Universal Robots PolyScope program: industrial_CHAIYO_TURBO.urp

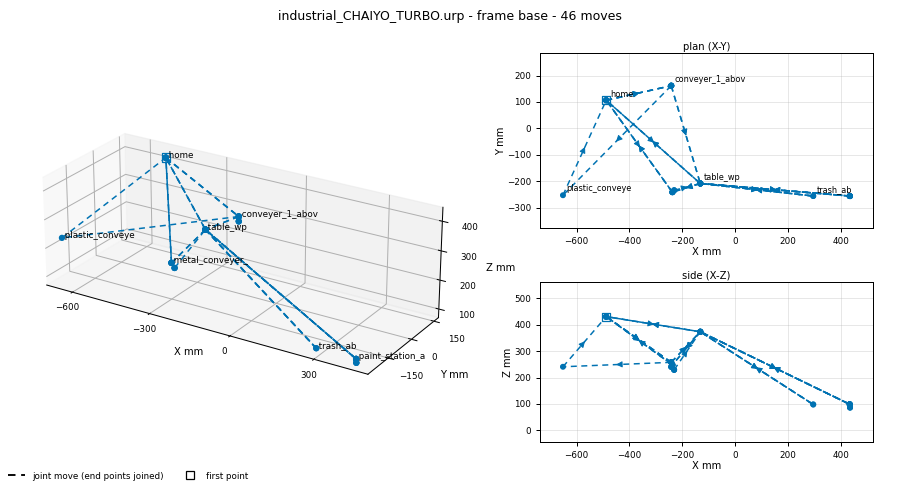
[picture p0: tool path of industrial_CHAIYO_TURBO.urp in frame base, 46 of 46 moves have a stored position in this frame; points joined in program order, loops and branches not executed]
Program industrial_CHAIYO_TURBO (createdIn=3.3.2.266 lastSavedIn=3.3.2.266 directory=/programs/usbdisk installation=default robotSerialNumber=2016353468)
Calibrated DH parameters: a=[0.000201, -0.204825, -0.377339, 0.000067, 0.000035, 0]; d=[0.089016, 277.403916, -258.203358, -19.0904, 0.094913, 0.082586]; alpha=[1.570161, 0.001342, -0.005575, 1.569994, -1.570842, 0]; deltaTheta=[0.000008, 1.067914, -1.344269, 0.276418, -0.000094, 0.00004]
Robot Program (runOnlyOnce=false motionType=MoveJ speed=1.047198 acceleration=1.396263 recalculateMotions=false)
  Set DigitalOutput pin=digital_out[4]; digitalValue=0
  var_1 := 0
  var_2 := 0
  var_3 := 0
  MoveJ speed 30 deg/s, acceleration 50 deg/s^2 (recalculateMotions=false)
    Waypoint home: TCP in base x=-488.151 y=106.291 z=430.627 mm, rx=1.1928 ry=2.9028 rz=-0.0084 rad; joints [180.494, -90.027, -89.995, -90.031, 90.023, -45] deg
  Wait DigitalInput pin=digital_in[0]; digitalValue=1
  If digital_in[1]
    var_1 := 1
  If digital_in[2]
    var_2 := 1
  If digital_in[3]
    var_3 := 1
  Set DigitalOutput pin=digital_out[0]; digitalValue=1
  Set DigitalOutput pin=digital_out[1]; digitalValue=1
  Switch expression=var_1*4+var_2*2+var_3*1
    Case (caseValue=1)
      MoveJ speed 50 deg/s, acceleration 60 deg/s^2 (recalculateMotions=false)
        Waypoint conveyer_1_abov: TCP in base x=-241.88 y=161.267 z=257.494 mm, rx=1.1929 ry=2.9028 rz=-0.0085 rad; joints [168.609, -62.296, -136.212, -71.617, 90.039, -56.942] deg
        Set DigitalOutput pin=digital_out[4]; digitalValue=1
      MoveJ speed 10 deg/s, acceleration 20 deg/s^2 (recalculateMotions=false)
        Waypoint conveyer_1: TCP in base x=-241.869 y=161.248 z=240.365 mm, rx=1.1929 ry=2.9028 rz=-0.0085 rad; joints [168.613, -63.476, -138.325, -68.325, 90.05, -56.955] deg
        Waypoint conveyer_1_abov: TCP in base x=-241.88 y=161.267 z=257.494 mm, rx=1.1929 ry=2.9028 rz=-0.0085 rad; joints [168.609, -62.296, -136.212, -71.617, 90.039, -56.942] deg
      MoveJ speed 50 deg/s, acceleration 60 deg/s^2 (recalculateMotions=false)
        Waypoint table_wp: motionParameters(blendRadius=0.05); TCP in base x=-131.8 y=-208.913 z=373.278 mm, rx=1.0433 ry=-2.9346 rz=0.1217 rad; joints [264.127, -50.382, -124.921, -90.048, 90.301, -45.115] deg
        Waypoint paint_station_a: TCP in base x=434.18 y=-256.504 z=98.644 mm, rx=-2.8837 ry=1.2374 rz=0.0692 rad; joints [342.112, -110.661, -119.501, -42.337, 90.247, -61.839] deg
      MoveJ speed 10 deg/s, acceleration 20 deg/s^2 (recalculateMotions=false)
        Waypoint paint_station: TCP in base x=435.467 y=-256.956 z=86.307 mm, rx=-2.883 ry=1.237 rz=0.0485 rad; joints [342.109, -112.325, -119.947, -39.471, 90.263, -61.851] deg
        Set DigitalOutput pin=digital_out[4]; digitalValue=0
      MoveJ speed 50 deg/s, acceleration 35 deg/s^2 (recalculateMotions=false)
        Waypoint paint_station_a: TCP in base x=434.18 y=-256.504 z=98.644 mm, rx=-2.8837 ry=1.2374 rz=0.0692 rad; joints [342.112, -110.661, -119.501, -42.337, 90.247, -61.839] deg
        Waypoint table_wp: motionParameters(blendRadius=0.05); TCP in base x=-131.8 y=-208.913 z=373.278 mm, rx=1.0433 ry=-2.9346 rz=0.1217 rad; joints [264.127, -50.382, -124.921, -90.048, 90.301, -45.115] deg
      Wait Sleep waitTime=7
      MoveJ speed 50 deg/s, acceleration 50 deg/s^2 (recalculateMotions=false)
        Waypoint table_wp: motionParameters(blendRadius=0.05); TCP in base x=-131.8 y=-208.913 z=373.278 mm, rx=1.0433 ry=-2.9346 rz=0.1217 rad; joints [264.127, -50.382, -124.921, -90.048, 90.301, -45.115] deg
        Waypoint paint_station_a: TCP in base x=434.18 y=-256.504 z=98.644 mm, rx=-2.8837 ry=1.2374 rz=0.0692 rad; joints [342.112, -110.661, -119.501, -42.337, 90.247, -61.839] deg
      Set DigitalOutput pin=digital_out[4]; digitalValue=1
      MoveJ speed 10 deg/s, acceleration 20 deg/s^2 (recalculateMotions=false)
        Waypoint paint_station: TCP in base x=435.467 y=-256.956 z=86.307 mm, rx=-2.883 ry=1.237 rz=0.0485 rad; joints [342.109, -112.325, -119.947, -39.471, 90.263, -61.851] deg
        Waypoint paint_station_a: TCP in base x=434.18 y=-256.504 z=98.644 mm, rx=-2.8837 ry=1.2374 rz=0.0692 rad; joints [342.112, -110.661, -119.501, -42.337, 90.247, -61.839] deg
      MoveJ speed 50 deg/s, acceleration 50 deg/s^2 (recalculateMotions=false)
        Waypoint table_wp: motionParameters(blendRadius=0.05); TCP in base x=-131.8 y=-208.913 z=373.278 mm, rx=1.0433 ry=-2.9346 rz=0.1217 rad; joints [264.127, -50.382, -124.921, -90.048, 90.301, -45.115] deg
        Waypoint metal_conveyer_: TCP in base x=-237.422 y=-242.02 z=247.737 mm, rx=1.1929 ry=2.9029 rz=-0.0083 rad; joints [244.594, -71.983, -132.548, -65.172, 89.926, 19.002] deg
      MoveJ speed 10 deg/s, acceleration 20 deg/s^2 (recalculateMotions=false)
        Waypoint metal_conveyer: TCP in base x=-230.831 y=-234.904 z=229.161 mm, rx=1.1929 ry=2.9028 rz=-0.0085 rad; joints [245.129, -71.78, -135.704, -62.218, 89.934, 19.525] deg
      Set DigitalOutput pin=digital_out[4]; digitalValue=0
      MoveJ speed 50 deg/s, acceleration 50 deg/s^2 (recalculateMotions=false)
        Waypoint metal_conveyer_: TCP in base x=-237.422 y=-242.02 z=247.737 mm, rx=1.1929 ry=2.9029 rz=-0.0083 rad; joints [244.594, -71.983, -132.548, -65.172, 89.926, 19.002] deg
        Waypoint home: TCP in base x=-488.151 y=106.291 z=430.627 mm, rx=1.1928 ry=2.9028 rz=-0.0084 rad; joints [180.494, -90.027, -89.995, -90.031, 90.023, -45] deg
    Case (caseValue=2)
      MoveJ speed 50 deg/s, acceleration 50 deg/s^2 (recalculateMotions=false)
        Waypoint table_wp: motionParameters(blendRadius=0.05); TCP in base x=-131.8 y=-208.913 z=373.278 mm, rx=1.0433 ry=-2.9346 rz=0.1217 rad; joints [264.127, -50.382, -124.921, -90.048, 90.301, -45.115] deg
        Waypoint paint_station_a: TCP in base x=434.18 y=-256.504 z=98.644 mm, rx=-2.8837 ry=1.2374 rz=0.0692 rad; joints [342.112, -110.661, -119.501, -42.337, 90.247, -61.839] deg
      Set DigitalOutput pin=digital_out[4]; digitalValue=1
      MoveJ speed 10 deg/s, acceleration 20 deg/s^2 (recalculateMotions=false)
        Waypoint paint_station: TCP in base x=435.467 y=-256.956 z=86.307 mm, rx=-2.883 ry=1.237 rz=0.0485 rad; joints [342.109, -112.325, -119.947, -39.471, 90.263, -61.851] deg
        Waypoint paint_station_a: TCP in base x=434.18 y=-256.504 z=98.644 mm, rx=-2.8837 ry=1.2374 rz=0.0692 rad; joints [342.112, -110.661, -119.501, -42.337, 90.247, -61.839] deg
      MoveJ speed 50 deg/s, acceleration 50 deg/s^2 (recalculateMotions=false)
        Waypoint table_wp: motionParameters(blendRadius=0.05); TCP in base x=-131.8 y=-208.913 z=373.278 mm, rx=1.0433 ry=-2.9346 rz=0.1217 rad; joints [264.127, -50.382, -124.921, -90.048, 90.301, -45.115] deg
        Waypoint metal_conveyer_: TCP in base x=-237.422 y=-242.02 z=247.737 mm, rx=1.1929 ry=2.9029 rz=-0.0083 rad; joints [244.594, -71.983, -132.548, -65.172, 89.926, 19.002] deg
      MoveJ speed 10 deg/s, acceleration 20 deg/s^2 (recalculateMotions=false)
        Waypoint metal_conveyer: TCP in base x=-230.831 y=-234.904 z=229.161 mm, rx=1.1929 ry=2.9028 rz=-0.0085 rad; joints [245.129, -71.78, -135.704, -62.218, 89.934, 19.525] deg
      Set DigitalOutput pin=digital_out[4]; digitalValue=0
      MoveJ speed 50 deg/s, acceleration 50 deg/s^2 (recalculateMotions=false)
        Waypoint metal_conveyer_: TCP in base x=-237.422 y=-242.02 z=247.737 mm, rx=1.1929 ry=2.9029 rz=-0.0083 rad; joints [244.594, -71.983, -132.548, -65.172, 89.926, 19.002] deg
        Waypoint home: TCP in base x=-488.151 y=106.291 z=430.627 mm, rx=1.1928 ry=2.9028 rz=-0.0084 rad; joints [180.494, -90.027, -89.995, -90.031, 90.023, -45] deg
    Case (caseValue=3)
      MoveJ speed 50 deg/s, acceleration 50 deg/s^2 (recalculateMotions=false)
        Waypoint conveyer_1_abov: TCP in base x=-241.88 y=161.267 z=257.494 mm, rx=1.1929 ry=2.9028 rz=-0.0085 rad; joints [168.609, -62.296, -136.212, -71.617, 90.039, -56.942] deg
      Set DigitalOutput pin=digital_out[4]; digitalValue=1
      MoveJ speed 5 deg/s, acceleration 20 deg/s^2 (recalculateMotions=false)
        Waypoint conveyer_1: TCP in base x=-241.869 y=161.248 z=240.365 mm, rx=1.1929 ry=2.9028 rz=-0.0085 rad; joints [168.613, -63.476, -138.325, -68.325, 90.05, -56.955] deg
        Waypoint conveyer_1_abov: TCP in base x=-241.88 y=161.267 z=257.494 mm, rx=1.1929 ry=2.9028 rz=-0.0085 rad; joints [168.609, -62.296, -136.212, -71.617, 90.039, -56.942] deg
      MoveJ speed 50 deg/s, acceleration 50 deg/s^2 (recalculateMotions=false)
        Waypoint plastic_conveye: TCP in base x=-651.975 y=-253.494 z=240.666 mm, rx=1.1928 ry=2.9027 rz=-0.0081 rad; joints [210.37, -121.891, -76.893, -71.085, 90.076, -15.248] deg; flange x=-651.997 y=-253.48 z=240.772 mm, rx=1.1928 ry=2.9028 rz=-0.0084 rad
      Set DigitalOutput pin=digital_out[4]; digitalValue=0
      MoveJ speed 50 deg/s, acceleration 50 deg/s^2 (recalculateMotions=false)
        Waypoint home: TCP in base x=-488.151 y=106.291 z=430.627 mm, rx=1.1928 ry=2.9028 rz=-0.0084 rad; joints [180.494, -90.027, -89.995, -90.031, 90.023, -45] deg
    Case (caseValue=4)
      MoveJ speed 50 deg/s, acceleration 50 deg/s^2 (recalculateMotions=false)
        Waypoint conveyer_1_abov: TCP in base x=-241.88 y=161.267 z=257.494 mm, rx=1.1929 ry=2.9028 rz=-0.0085 rad; joints [168.609, -62.296, -136.212, -71.617, 90.039, -56.942] deg
      Set DigitalOutput pin=digital_out[4]; digitalValue=1
      MoveJ speed 10 deg/s, acceleration 20 deg/s^2 (recalculateMotions=false)
        Waypoint conveyer_1: TCP in base x=-241.869 y=161.248 z=240.365 mm, rx=1.1929 ry=2.9028 rz=-0.0085 rad; joints [168.613, -63.476, -138.325, -68.325, 90.05, -56.955] deg
        Waypoint conveyer_1_abov: TCP in base x=-241.88 y=161.267 z=257.494 mm, rx=1.1929 ry=2.9028 rz=-0.0085 rad; joints [168.609, -62.296, -136.212, -71.617, 90.039, -56.942] deg
      MoveJ speed 50 deg/s, acceleration 50 deg/s^2 (recalculateMotions=false)
        Waypoint table_wp: motionParameters(blendRadius=0.05); TCP in base x=-131.8 y=-208.913 z=373.278 mm, rx=1.0433 ry=-2.9346 rz=0.1217 rad; joints [264.127, -50.382, -124.921, -90.048, 90.301, -45.115] deg
        Waypoint trash_ab: TCP in base x=296.081 y=-256.486 z=97.854 mm, rx=-2.8837 ry=1.2373 rz=0.0692 rad; joints [335.557, -98.721, -137.069, -36.736, 89.977, -68.389] deg
      Set DigitalOutput pin=digital_out[4]; digitalValue=0
      MoveJ speed 50 deg/s, acceleration 50 deg/s^2 (recalculateMotions=false)
        Waypoint table_wp: motionParameters(blendRadius=0.05); TCP in base x=-131.8 y=-208.913 z=373.278 mm, rx=1.0433 ry=-2.9346 rz=0.1217 rad; joints [264.127, -50.382, -124.921, -90.048, 90.301, -45.115] deg
        Waypoint home: TCP in base x=-488.151 y=106.291 z=430.627 mm, rx=1.1928 ry=2.9028 rz=-0.0084 rad; joints [180.494, -90.027, -89.995, -90.031, 90.023, -45] deg
    Case (caseValue=5)
      MoveJ speed 50 deg/s, acceleration 50 deg/s^2 (recalculateMotions=false)
        Waypoint metal_conveyer_: TCP in base x=-237.422 y=-242.02 z=247.737 mm, rx=1.1929 ry=2.9029 rz=-0.0083 rad; joints [244.594, -71.983, -132.548, -65.172, 89.926, 19.002] deg
      Set DigitalOutput pin=digital_out[4]; digitalValue=1
      MoveJ speed 10 deg/s, acceleration 20 deg/s^2 (recalculateMotions=false)
        Waypoint metal_conveyer: TCP in base x=-230.831 y=-234.904 z=229.161 mm, rx=1.1929 ry=2.9028 rz=-0.0085 rad; joints [245.129, -71.78, -135.704, -62.218, 89.934, 19.525] deg
      MoveJ speed 50 deg/s, acceleration 50 deg/s^2 (recalculateMotions=false)
        Waypoint table_wp: motionParameters(blendRadius=0.05); TCP in base x=-131.8 y=-208.913 z=373.278 mm, rx=1.0433 ry=-2.9346 rz=0.1217 rad; joints [264.127, -50.382, -124.921, -90.048, 90.301, -45.115] deg
        Waypoint trash_ab: TCP in base x=296.081 y=-256.486 z=97.854 mm, rx=-2.8837 ry=1.2373 rz=0.0692 rad; joints [335.557, -98.721, -137.069, -36.736, 89.977, -68.389] deg
      Set DigitalOutput pin=digital_out[4]; digitalValue=0
      MoveJ speed 50 deg/s, acceleration 50 deg/s^2 (recalculateMotions=false)
        Waypoint table_wp: motionParameters(blendRadius=0.05); TCP in base x=-131.8 y=-208.913 z=373.278 mm, rx=1.0433 ry=-2.9346 rz=0.1217 rad; joints [264.127, -50.382, -124.921, -90.048, 90.301, -45.115] deg
        Waypoint home: TCP in base x=-488.151 y=106.291 z=430.627 mm, rx=1.1928 ry=2.9028 rz=-0.0084 rad; joints [180.494, -90.027, -89.995, -90.031, 90.023, -45] deg
    Case (caseValue=2147483647)
      Set DigitalOutput pin=digital_out[4]; digitalValue=0
      MoveJ speed 50 deg/s, acceleration 30 deg/s^2 (recalculateMotions=false)
        Waypoint home: TCP in base x=-488.151 y=106.291 z=430.627 mm, rx=1.1928 ry=2.9028 rz=-0.0084 rad; joints [180.494, -90.027, -89.995, -90.031, 90.023, -45] deg
  Set DigitalOutput pin=digital_out[0]; digitalValue=0
  Set DigitalOutput pin=digital_out[1]; digitalValue=0
  Script: sync()
  SuppressedNode
    MoveJ speed 60 deg/s, acceleration 80 deg/s^2 (recalculateMotions=false)
      Waypoint conveyer_1: TCP in base x=-241.882 y=161.249 z=240.765 mm, rx=1.1928 ry=2.9027 rz=-0.0085 rad; joints [168.613, -63.44, -138.267, -68.419, 90.049, -56.954] deg; flange x=-241.871 y=161.257 z=240.815 mm, rx=1.1928 ry=2.9028 rz=-0.0084 rad
      Waypoint conveyer_1_abov: TCP in base x=-241.88 y=161.267 z=257.494 mm, rx=1.1929 ry=2.9028 rz=-0.0085 rad; joints [168.609, -62.296, -136.212, -71.617, 90.039, -56.942] deg
      Waypoint metal_conveyer: TCP in base x=-246.394 y=-211.361 z=228.562 mm, rx=1.1928 ry=2.9028 rz=-0.0083 rad; joints [240.54, -70.976, -136.281, -62.461, 89.956, 14.938] deg
      Waypoint metal_conveyer_: TCP in base x=-246.409 y=-211.393 z=242.589 mm, rx=1.1929 ry=2.9028 rz=-0.0084 rad; joints [240.537, -69.797, -134.708, -65.213, 89.946, 14.948] deg
      Waypoint table_wp: TCP in base x=-131.8 y=-208.913 z=373.278 mm, rx=1.0433 ry=-2.9346 rz=0.1217 rad; joints [264.127, -50.382, -124.921, -90.048, 90.301, -45.115] deg
      Waypoint paint_station: TCP in base x=441.254 y=-256.466 z=85.146 mm, rx=-2.8835 ry=1.2373 rz=0.0692 rad; joints [342.362, -112.888, -118.985, -40.624, 90.268, -61.596] deg; flange x=441.235 y=-256.498 z=85.182 mm, rx=-2.8837 ry=1.2374 rz=0.0691 rad
      Waypoint paint_station_a: TCP in base x=441.257 y=-256.487 z=98.666 mm, rx=-2.8837 ry=1.2373 rz=0.069 rad; joints [342.36, -111.279, -118.512, -42.707, 90.256, -61.591] deg
      Waypoint trash_ab: TCP in base x=296.081 y=-256.486 z=97.854 mm, rx=-2.8837 ry=1.2373 rz=0.0692 rad; joints [335.557, -98.721, -137.069, -36.736, 89.977, -68.389] deg
      Waypoint trash: TCP in base x=296.062 y=-256.514 z=85.005 mm, rx=-2.8837 ry=1.2374 rz=0.0692 rad; joints [335.56, -100.877, -137.652, -33.997, 89.994, -68.394] deg
      Waypoint plastic_conveye: TCP in base x=-651.975 y=-253.494 z=240.666 mm, rx=1.1928 ry=2.9027 rz=-0.0081 rad; joints [210.37, -121.891, -76.893, -71.085, 90.076, -15.248] deg; flange x=-651.997 y=-253.48 z=240.772 mm, rx=1.1928 ry=2.9028 rz=-0.0084 rad
